// TIA Portal V17 export
// export: Created 2023-12-22T15:03:17.8188599Z, ExportSetting WithDefaults, DisplayName Totally Integrated Automation Portal, DisplayVersion V17, DisplayName TIA Portal Openness, DisplayVersion V17, DisplayName TIA Portal Version Control Interface, DisplayVersion V17, DisplayName STEP 7 Professional, DisplayVersion V17, DisplayName STEP 7 Safety, DisplayVersion V17, DisplayName WinCC Advanced, DisplayVersion V17
DATA_BLOCK "SKV_cnt_DB"   // DB4
VERSION : 0.1
// stored: AutoNumber true, DBAccessibleFromOPCUA true, DBAccessibleFromWebserver true, InstanceOfName SKV_cnt, InstanceOfType FB
"SKV_cnt"
   // VAR RETAIN
   //    CMD : Struct
   //       Select : Bool;
   //       Mode : Bool;
   //       Rotation : Bool;
   //       Load : Bool;
   //       Reload : Bool;
   //       Deload : Bool;
   //       Add : Bool;
   //       REQ : Int;
   //    END_STRUCT;
   //    Data : Struct
   //       Ready : Bool;
   //       Add_Ready : Bool;
   //       C : Real;
   //       REQ : Int;
   //       N : Int;
   //       Status : Int;
   //       N_On : Int;
   //       N_Off : Int;
   //    END_STRUCT;
   //    "Step" : Int;
   //    dev : Int;
   //    Clock { S7_SetPoint := 'True'} : Array[0..4] of "Time_S";
   // END_VAR
BEGIN
   Clock[0].SP := 10;
   Clock[1..4].SP := 2;
END_DATA_BLOCK
